// TwinCAT 3 PLC project PLC_Tank
// ProgramVersion: 3.1.4024.0
// libraries:
//   Tc2_ControllerToolbox, * (Beckhoff Automation GmbH)
//   Tc2_ModbusSrv, * (Beckhoff Automation GmbH)
//   Tc2_Standard, * (Beckhoff Automation GmbH)
//   Tc2_System, * (Beckhoff Automation GmbH)
//   Tc3_Module, * (Beckhoff Automation GmbH)
//   VisuDialogs, * (System)
//   VisuSymbols,3.5.10.0,System
// project tree:
//   DUTs/ TAnalogConversion.TcDUT, TEngine.TcDUT, TEngineCmd.TcDUT, THeaterState.TcDUT, THeaterCmd.TcDUT, THeater.TcDUT, TPhaseHeating.TcDUT, TPhaseCmd.TcDUT, TPhaseDraining.TcDUT, TPhaseFilling.TcDUT, TPhaseMixing.TcDUT, TPhaseState.TcDUT, TValveState.TcDUT, TValveCmd.TcDUT, TEngineState.TcDUT, TTank.TcDUT, TValve.TcDUT
//   / GlobalTextList.TcGTLO, PlcTask.TcTTO, PlcTask500ms.TcTTO, Visualization Manager.TcVMO (not stored)
//   GVLs/ Global.TcGVL
//   POUs/ Draining.TcPOU, Engine_1DO.TcPOU, FB_Tank.TcPOU, Filling.TcPOU, Heater.TcPOU, Heating.TcPOU, Main_Batch.TcPOU, MB_Connector.TcPOU, Mixing.TcPOU, Test.TcPOU, Valve_2DO.TcPOU, MAIN.TcPOU
//   POUs/Misc/ EngToRaw.TcPOU, RawToEng.TcPOU
//   VISUs/ Visualization.TcVIS
// real-time tasks:
//   TASK PlcTask: cycle T#100000us, priority 20, ADS port 350
//   TASK PlcTask500ms: cycle T#500ms, priority 1, ADS port 351

CONFIGURATION PLC_Tank
    RESOURCE PLC ON TwinCAT3
        TASK PlcTask(INTERVAL := T#100000us, PRIORITY := 20);
        TASK PlcTask500ms(INTERVAL := T#500ms, PRIORITY := 1);
        PROGRAM MB_Connector WITH PlcTask : MB_Connector;
        PROGRAM Main_Batch WITH PlcTask : Main_Batch;
        PROGRAM MAIN WITH PlcTask500ms : MAIN;
    END_RESOURCE
END_CONFIGURATION

// ---- DUTs/TAnalogConversion.TcDUT
TYPE TAnalogConversion :
STRUCT
	TransducerLoLevel : UINT;
	TransducerHiLevel : UINT;
	ScaledValLoLevel : REAL;
	ScaledValHiLevel : REAL;
END_STRUCT
END_TYPE

// ---- DUTs/TEngine.TcDUT
TYPE TEngine :
STRUCT
	Cmd : TEngineCmd;
	State : TEngineState;
	Time2Start : TIME := T#5S;
	RisingEdgeTrigger : R_TRIG;
	StartupFailTimer : TON;
END_STRUCT
END_TYPE

// ---- DUTs/TEngineCmd.TcDUT
TYPE TEngineCmd :
STRUCT
		SetRT : DINT;
		AutCtrl : BOOL;
		ManCtrl : BOOL;
		TurnOnMan : BOOL;
		TurnOffMan : BOOL;
		Req2RunAutCtrl : BOOL;
		ResetSUF : BOOL;
END_STRUCT
END_TYPE

// ---- DUTs/THeaterState.TcDUT
TYPE THeaterState :
STRUCT
	EnableOut : BOOL;
	HeatingOut : REAL;
	AutCtrl : BOOL;
	ManCtrl : BOOL;
	Err 	: BOOL;
	StateInt : INT;
	GenErr : BOOL; //signalisation: error occured

	HeatingPower : REAL;
	

END_STRUCT
END_TYPE

// ---- DUTs/THeaterCmd.TcDUT
TYPE THeaterCmd :
STRUCT
	AutCtrl : BOOL;
	ManCtrl : BOOL;
	TurnOnMan : BOOL;
	TurnOffMan : BOOL;
	Req2RunAutCtrl : BOOL;
END_STRUCT
END_TYPE

// ---- DUTs/THeater.TcDUT
TYPE THeater :
STRUCT
	Cmd : THeaterCmd;
	State : THeaterState;
	
	ParamHeatingPowerManual : REAL;
	ParamHeatingSetPointAutomat : REAL;
	
	PID : FB_CTRL_PID;
	ThresholdTimer : TON;
	
END_STRUCT
END_TYPE

// ---- DUTs/TPhaseHeating.TcDUT
TYPE TPhaseHeating :
STRUCT
	Cmd : TPhaseCmd;
	State : TPhaseState;
	
	ParamReqTemp : REAL;
	
	WaterTemp : REAL;
	
	fTime : INT;
END_STRUCT
END_TYPE

// ---- DUTs/TPhaseCmd.TcDUT
TYPE TPhaseCmd :
STRUCT
	StartAut : BOOL;
	StopAut : BOOL;
	StartMan : BOOL;
	StopMan : BOOL;
	PauseMan : BOOL;
	ResumeMan : BOOL;
	ResetDone : BOOL;
	AutCtrl : BOOL;
	ManCtrl : BOOL;
END_STRUCT
END_TYPE

// ---- DUTs/TPhaseDraining.TcDUT
TYPE TPhaseDraining :
STRUCT
	Cmd : TPhaseCmd;
	State : TPhaseState;
	
	ParamDrainLevel : REAL;
	WaterLevel : REAL;
END_STRUCT
END_TYPE

// ---- DUTs/TPhaseFilling.TcDUT
TYPE TPhaseFilling :
STRUCT
	Cmd : TPhaseCmd;
	State : TPhaseState;
	
	ParamFillLevel : REAL;
	WaterLevel : REAL;
END_STRUCT
END_TYPE

// ---- DUTs/TPhaseMixing.TcDUT
TYPE TPhaseMixing :
STRUCT
	Cmd : TPhaseCmd;
	State : TPhaseState;
	
	ParamTimeSec : INT;
	
	ElapsedTimeSec : INT;
END_STRUCT
END_TYPE

// ---- DUTs/TPhaseState.TcDUT
TYPE TPhaseState :
STRUCT
	Running : BOOL;
	Idle : BOOL;
	Paused : BOOL;
	Done : BOOL;
	AutCtrl : BOOL;
	ManCtrl : BOOL;
	Stateint : INT;
END_STRUCT
END_TYPE

// ---- DUTs/TValveState.TcDUT
TYPE TValveState :
STRUCT
		Open : BOOL;
		Closed : BOOL;
		OpenOut : BOOL;
		CloseOut : BOOL;
		Err : BOOL;
		StartupFail : BOOL;
		AutCtrl : BOOL;
		ManCtrl : BOOL;
		MayRun : BOOL;
		MayAutoRun : BOOL; //device is working in automatic regime
		GenErr : BOOL; //signalisation: error occured
		StColor : INT; //valve state: Open(0), Closed(1), OpenAndErr(2), ClosedAndErr(3) ,NotOpenNotClosedNotErr(4), NotOpenNotClosedAndErr(5), OpenAndClosedAndErr(6), OpenAndClosedNotErr(7)

END_STRUCT
END_TYPE

// ---- DUTs/TValveCmd.TcDUT
TYPE TValveCmd :
STRUCT
		AutCtrl : BOOL;
		ManCtrl : BOOL;
		OpenMan : BOOL;
		StopMan : BOOL;
		CloseMan : BOOL;
		Req2OpenAut : BOOL;
		Req2CloseAut : BOOL;
		ResetSUF : BOOL;
END_STRUCT
END_TYPE

// ---- DUTs/TEngineState.TcDUT
TYPE TEngineState :
STRUCT
		RT : DINT;
		Run : BOOL;
		RunOut : BOOL;
		Err : BOOL;
		StartUpFail : BOOL;
		AutCtrl : BOOL;
		ManCtrl : BOOL;
		MayRun : BOOL;
		MayAutoRun : BOOL;
		GenErr : BOOL;
		StateInt : INT;
		
		StartupFailTime : INT;
END_STRUCT
END_TYPE

// ---- DUTs/TTank.TcDUT
TYPE TTank :
STRUCT
	Mixer : TEngine;
	ValveFilling : TValve;
	ValveDraining : TValve;
	Heater : THeater;
	
	Filling : TPhaseFilling;
	Draining : TPhaseDraining;
	Mixing : TPhaseMixing;
	Heating : TPhaseHeating;
	
	GlobalError : BOOL;

END_STRUCT
END_TYPE

// ---- DUTs/TValve.TcDUT
TYPE TValve :
STRUCT
	Cmd : TValveCmd;
	State : TValveState;
	Time2Open : TIME := T#12S;
	
	OpenFailTimer : TON;
	CloseFailTimer : TON;
	
END_STRUCT
END_TYPE

// ---- GVLs/Global.TcGVL
{attribute 'qualified_only'}
VAR_GLOBAL
	Tank1 : TTank;
	

	secImp : BOOL;
	
	diMixerRun : BOOL;
	diMixerError : BOOL;
	diValveFillOpen : BOOL;
	diValveFillClose : BOOL;
	diValveFillError : BOOL;
	diValveDrainOpen : BOOL;
	diValveDrainClose : BOOL;
	diValveDrainError : BOOL;
	
	aiWaterLevel : WORD;
	aiWaterTemp : WORD;
	
	doMixerStart : BOOL;
	doValveFillOpen : BOOL;
	doValveFillClose : BOOL;
	doValveDrainOpen : BOOL;
	doValveDrainClose : BOOL;
	doHeatingEnable : BOOL;
	
	aoReqPowerOfHeating : WORD;

END_VAR

VAR_GLOBAL CONSTANT
	Running : INT := 0;
	Stop : INT := 1;
	RunningAndError : INT := 2;
	Err : INT := 3;

	PhIdle : INT := 0;
	PhRunning : INT := 1;
	PhPause : INT := 2;
	
    Open : INT := 0;
	Closed : INT := 1;
	OpenAndErr : INT := 2;
	ClosedAndErr : INT := 3;
	NotOpenNotClosedNotErr : INT := 4;
	NotOpenNotClosedAndErr : INT := 5;
	OpenAndClosedAndErr : INT := 6;
	OpenAndClosedNotErr : INT := 7;
END_VAR

// ---- POUs/MB_Connector.TcPOU
PROGRAM MB_Connector
VAR
	
	mb_ipaddr   : STRING(15) := '127.0.0.1';
	mb_port		: UINT := 503;
	mb_unitid	: BYTE := 1;
	
	fbReadRegs		: FB_MBReadInputRegs;
	mb_regs    		: ARRAY [0..4] OF WORD;
	mb_regs_error	: BOOL;
	mb_regs_busy	: BOOL;
	mb_regs_execute : BOOL;
	mb_regs_errid	: UDINT;
	
	fbReadInps	: FB_MBReadInputs;
	mb_inps			: ARRAY [0..4] OF BYTE;
	mb_inps_error	: BOOL;
	mb_inps_busy	: BOOL;
	mb_inps_execute : BOOL;
	mb_inps_errid	: UDINT;
	
	fbWriteRegs		: FB_MBWriteRegs;
	mbw_regs    	: ARRAY [0..4] OF WORD;
	mbw_regs_error	: BOOL;
	mbw_regs_busy	: BOOL;
	mbw_regs_execute: BOOL;
	mbw_regs_errid	: UDINT;
	
	fbWriteCoils	: FB_MBWriteCoils;
	mbw_coils		: ARRAY [0..4] OF BYTE;
	mbw_coils_error	: BOOL;
	mbw_coils_busy	: BOOL;
	mbw_coils_execute: BOOL;
	mbw_coils_errid	: UDINT;
	
END_VAR

fbReadRegs.sIPAddr := mb_ipaddr;
fbReadRegs.nTCPPort := mb_port;
fbReadRegs.nQuantity := 4;
fbReadRegs.nMBAddr := 0;
fbReadRegs.cbLength := SIZEOF(mb_regs);
fbReadRegs.pDestAddr := ADR(mb_regs);
fbReadRegs.nUnitID := mb_unitid;
fbReadRegs.tTimeout := T#5S;
IF (mb_regs_busy = FALSE) THEN
	mb_regs_execute := TRUE;
ELSE
	mb_regs_execute := FALSE;
END_IF
fbReadRegs(bExecute := mb_regs_execute, 
		   bBusy => mb_regs_busy, bError => mb_regs_error, 
		   nErrId => mb_regs_errid);



fbReadInps.sIPAddr := mb_ipaddr;
fbReadInps.nTCPPort := mb_port;
fbReadInps.nQuantity := 32;
fbReadInps.nMBAddr := 0;
fbReadInps.cbLength := SIZEOF(mb_inps);
fbReadInps.pDestAddr := ADR(mb_inps);
fbReadInps.nUnitID := mb_unitid;
fbReadInps.tTimeout := T#5S;
IF (mb_inps_busy = FALSE) THEN
	mb_inps_execute := TRUE;
ELSE
	mb_inps_execute := FALSE;
END_IF
fbReadInps(bExecute := mb_inps_execute, 
	bBusy => mb_inps_busy, bError => mb_inps_error, nErrId => mb_inps_errid);

Global.diValveFillOpen := mb_inps[0].0;
Global.diValveFillClose := mb_inps[0].1;
Global.diValveFillError := mb_inps[0].2;
Global.diValveDrainOpen := mb_inps[0].3;
Global.diValveDrainClose := mb_inps[0].4;
Global.diValveDrainError := mb_inps[0].5;
Global.diMixerRun := mb_inps[0].6;
Global.diMixerError := mb_inps[0].7;

Global.aiWaterLevel := mb_regs[0];
Global.aiWaterTemp := mb_regs[2];







fbWriteRegs.sIPAddr := mb_ipaddr;
fbWriteRegs.nTCPPort := mb_port;
fbWriteRegs.nQuantity := 4;
fbWriteRegs.nMBAddr := 0;
fbWriteRegs.cbLength := SIZEOF(mbw_regs);
fbWriteRegs.pSrcAddr := ADR(mbw_regs);
fbWriteRegs.nUnitID := mb_unitid;
fbWriteRegs.tTimeout := T#5S;
IF (mbw_regs_busy = FALSE) THEN
	mbw_regs_execute := TRUE;
ELSE
	mbw_regs_execute := FALSE;
END_IF
fbWriteRegs(bExecute := mbw_regs_execute, 
		   bBusy => mbw_regs_busy, bError => mbw_regs_error, 
		   nErrId => mbw_regs_errid);



fbWriteCoils.sIPAddr := mb_ipaddr;
fbWriteCoils.nTCPPort := mb_port;
fbWriteCoils.nQuantity := 32;
fbWriteCoils.nMBAddr := 0;
fbWriteCoils.cbLength := SIZEOF(mbw_coils);
fbWriteCoils.pSrcAddr := ADR(mbw_coils);
fbWriteCoils.nUnitID := mb_unitid;
fbWriteCoils.tTimeout := T#5S;
IF (mbw_coils_busy = FALSE) THEN
	mbw_coils_execute := TRUE;
ELSE
	mbw_coils_execute := FALSE;
END_IF
fbWriteCoils(bExecute := mbw_coils_execute, 
	bBusy => mbw_coils_busy, bError => mbw_coils_error, nErrId => mbw_coils_errid);

mbw_coils[0].0 := Global.doValveFillOpen;
mbw_coils[0].1 := Global.doValveFillClose;
mbw_coils[0].2 := Global.doValveDrainOpen;
mbw_coils[0].3 := Global.doValveDrainClose;
mbw_coils[0].4 := Global.doMixerStart;
mbw_coils[0].5 := Global.doHeatingEnable;

mbw_regs[0] := Global.aoReqPowerOfHeating;

END_PROGRAM

// ---- POUs/Main_Batch.TcPOU
PROGRAM Main_Batch
VAR
	FB_Tank_1 : FB_Tank;
END_VAR

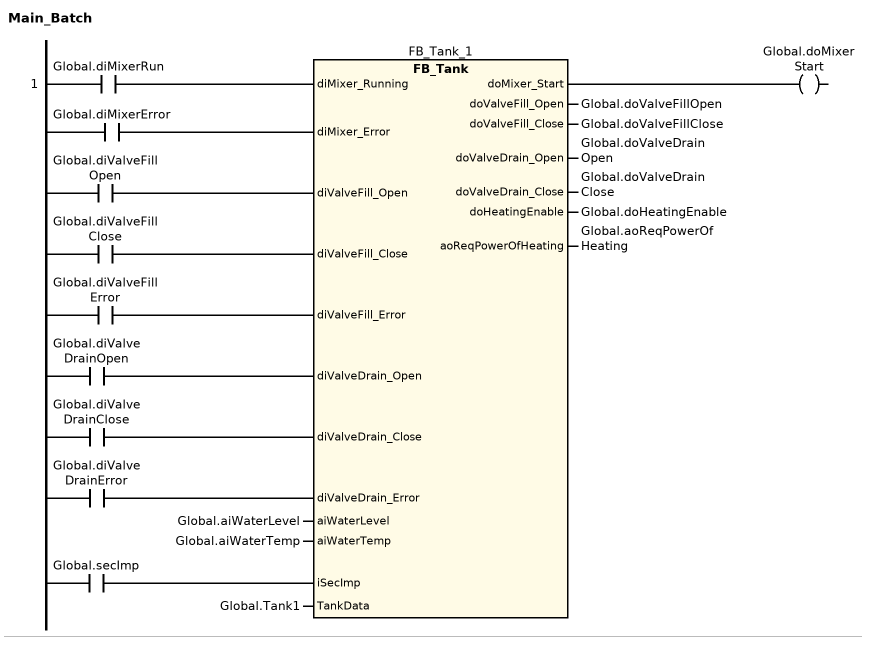
// NETWORK 1
FB_Tank_1(
    diMixer_Running := Global.diMixerRun,
    diMixer_Error := Global.diMixerError,
    diValveFill_Open := Global.diValveFillOpen,
    diValveFill_Close := Global.diValveFillClose,
    diValveFill_Error := Global.diValveFillError,
    diValveDrain_Open := Global.diValveDrainOpen,
    diValveDrain_Close := Global.diValveDrainClose,
    diValveDrain_Error := Global.diValveDrainError,
    aiWaterLevel := Global.aiWaterLevel,
    aiWaterTemp := Global.aiWaterTemp,
    iSecImp := Global.secImp,
    TankData := Global.Tank1,
    doValveFill_Open => Global.doValveFillOpen,
    doValveFill_Close => Global.doValveFillClose,
    doValveDrain_Open => Global.doValveDrainOpen,
    doValveDrain_Close => Global.doValveDrainClose,
    doHeatingEnable => Global.doHeatingEnable,
    aoReqPowerOfHeating => Global.aoReqPowerOfHeating); // FB_Tank
Global.doMixerStart := FB_Tank_1.doMixer_Start;

END_PROGRAM

// ---- POUs/FB_Tank.TcPOU
FUNCTION_BLOCK FB_Tank
VAR_INPUT
	diMixer_Running : BOOL;
	diMixer_Error : BOOL;
	diValveFill_Open : BOOL;
	diValveFill_Close : BOOL;
	diValveFill_Error : BOOL;
	diValveDrain_Open : BOOL;
	diValveDrain_Close : BOOL;
	diValveDrain_Error : BOOL;
	aiWaterLevel : WORD;
	aiWaterTemp : WORD;
	iSecImp : BOOL; //Požaduje se vstup s periodou 1 sekunda a libovolnou střídou
END_VAR

VAR_OUTPUT
	doMixer_Start : BOOL;
	doValveFill_Open : BOOL;
	doValveFill_Close : BOOL;
	doValveDrain_Open : BOOL;
	doValveDrain_Close : BOOL;
	doHeatingEnable : BOOL;
	aoReqPowerOfHeating : WORD;
END_VAR

VAR_IN_OUT
	TankData : TTank;
END_VAR

VAR
	//Konfigurace přepočtu rozsahu převodníků
	WaterTemp : TAnalogConversion := (TransducerLoLevel := 0, TransducerHiLevel := 27648, ScaledValLoLevel := 0, ScaledValHiLevel := 100);
	WaterLevel : TAnalogConversion := (TransducerLoLevel := 0, TransducerHiLevel := 27648, ScaledValLoLevel := 0, ScaledValHiLevel := 2);
	ReqOutputPower : TAnalogConversion := (ScaledValLoLevel := 0, ScaledValHiLevel := 100, TransducerLoLevel := 0, TransducerHiLevel := 27648);

	//Instance zanořených funkčních bloků
	ValveDrainCm : Valve_2DO;
	ValveFillCm : Valve_2DO;
	MixerCm : Engine_1DO;
	HeaterCm : Heater;
	FillingPhase : Filling;
	MixingPhase : Mixing;
	DrainingPhase : Draining;
	HeatingPhase : Heating;
	TON1: TON;
	RawToEng_1: RawToEng;
	RawToEng_2: RawToEng;
	EngToRaw_1: EngToRaw;
END_VAR

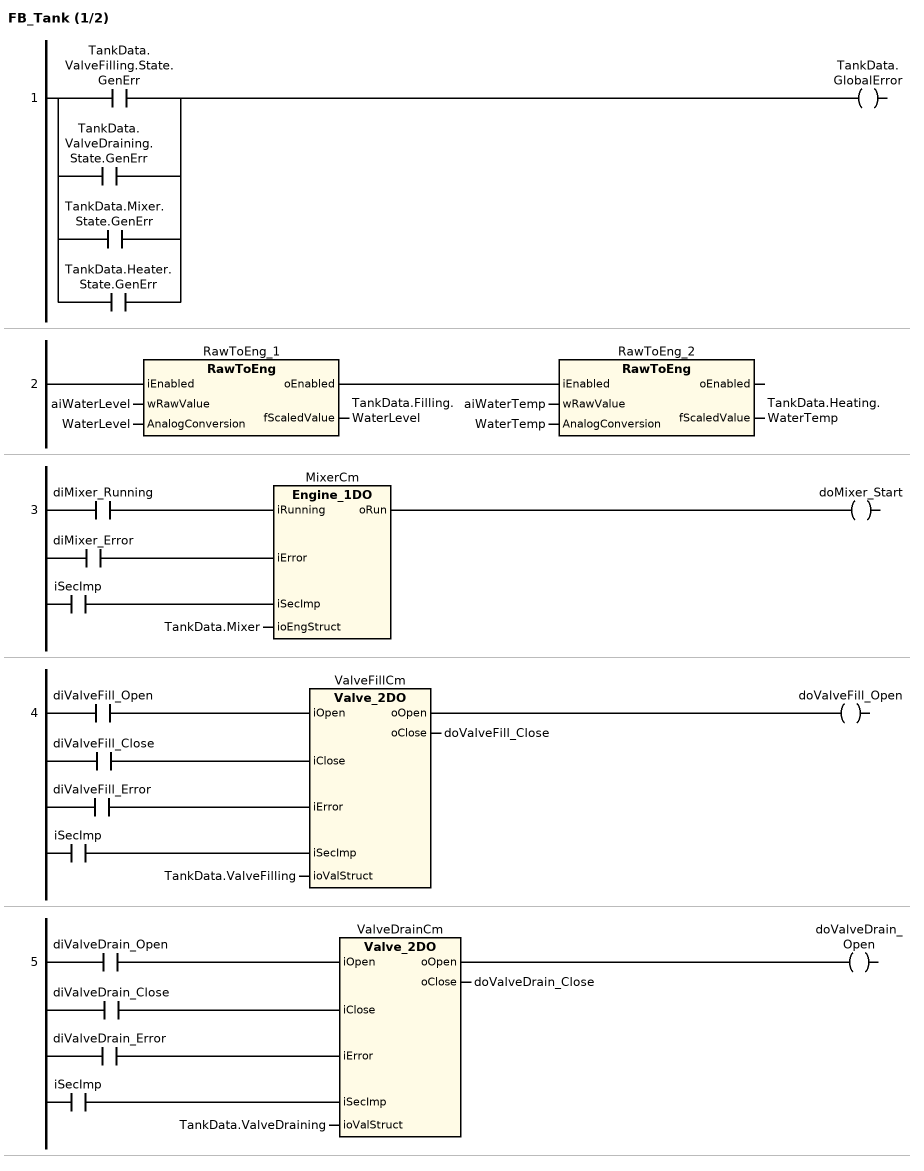
// NETWORK 1
TankData.GlobalError := TankData.ValveFilling.State.GenErr OR TankData.ValveDraining.State.GenErr OR TankData.Mixer.State.GenErr OR TankData.Heater.State.GenErr;

// NETWORK 2
RawToEng_1(
    iEnabled := TRUE,
    wRawValue := aiWaterLevel,
    AnalogConversion := WaterLevel,
    fScaledValue => TankData.Filling.WaterLevel); // RawToEng
RawToEng_2(
    iEnabled := RawToEng_1.oEnabled,
    wRawValue := aiWaterTemp,
    AnalogConversion := WaterTemp,
    fScaledValue => TankData.Heating.WaterTemp); // RawToEng

// NETWORK 3
MixerCm(
    iRunning := diMixer_Running,
    iError := diMixer_Error,
    iSecImp := iSecImp,
    ioEngStruct := TankData.Mixer); // Engine_1DO
doMixer_Start := MixerCm.oRun;

// NETWORK 4
ValveFillCm(
    iOpen := diValveFill_Open,
    iClose := diValveFill_Close,
    iError := diValveFill_Error,
    iSecImp := iSecImp,
    ioValStruct := TankData.ValveFilling,
    oClose => doValveFill_Close); // Valve_2DO
doValveFill_Open := ValveFillCm.oOpen;

// NETWORK 5
ValveDrainCm(
    iOpen := diValveDrain_Open,
    iClose := diValveDrain_Close,
    iError := diValveDrain_Error,
    iSecImp := iSecImp,
    ioValStruct := TankData.ValveDraining,
    oClose => doValveDrain_Close); // Valve_2DO
doValveDrain_Open := ValveDrainCm.oOpen;

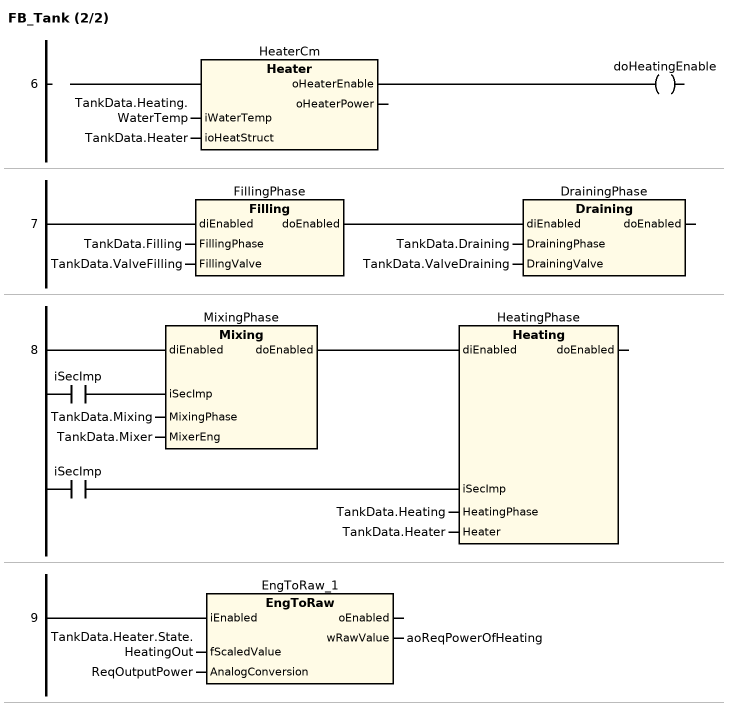
// NETWORK 6
HeaterCm(iWaterTemp := TankData.Heating.WaterTemp, ioHeatStruct := TankData.Heater); // Heater
doHeatingEnable := HeaterCm.oHeaterEnable;

// NETWORK 7
FillingPhase(diEnabled := TRUE, FillingPhase := TankData.Filling, FillingValve := TankData.ValveFilling); // Filling
DrainingPhase(
    diEnabled := FillingPhase.doEnabled,
    DrainingPhase := TankData.Draining,
    DrainingValve := TankData.ValveDraining); // Draining

// NETWORK 8
MixingPhase(
    diEnabled := TRUE,
    iSecImp := iSecImp,
    MixingPhase := TankData.Mixing,
    MixerEng := TankData.Mixer); // Mixing
HeatingPhase(
    diEnabled := MixingPhase.doEnabled,
    iSecImp := iSecImp,
    HeatingPhase := TankData.Heating,
    Heater := TankData.Heater); // Heating

// NETWORK 9
EngToRaw_1(
    iEnabled := TRUE,
    fScaledValue := TankData.Heater.State.HeatingOut,
    AnalogConversion := ReqOutputPower,
    wRawValue => aoReqPowerOfHeating); // EngToRaw

END_FUNCTION_BLOCK

// ---- POUs/Valve_2DO.TcPOU
FUNCTION_BLOCK Valve_2DO
VAR_INPUT
	iOpen : BOOL;
	iClose : BOOL;
	iError : BOOL;
	iSecImp : BOOL;
END_VAR
VAR_OUTPUT
	oOpen : BOOL;
	oClose : BOOL;
END_VAR

VAR_IN_OUT
	ioValStruct	 : TValve;
END_VAR

VAR
	tempOpenStartupFail : BOOL;
	tempCloseStartupFail: BOOL;
END_VAR

{region "OpenState"}
    // set real state of valve input into valve structure - input of valve can be taken from limit sensor...
    ioValStruct.State.Open := iOpen;
    ioValStruct.State.Closed := iClose;
{endregion}

	 
{region "Manual/Automat"}
	// switching state of engine - automatic or manual control (default state is manual)
	
{endregion}
	 
{region "MayRun / MayAutoRun"}
    // setting auxilary signals (may run, may auto run) - MR AND NOT MAR - engine may be started in manual mode, MAR - engine may be started in automatic mode
    ioValStruct.State.MayRun := (ioValStruct.State.ManCtrl AND NOT(ioValStruct.State.GenErr));
	ioValStruct.State.MayAutoRun := (ioValStruct.State.AutCtrl AND NOT(ioValStruct.State.GenErr));
{endregion}
	 
{region "ManCtrl"}
	// processing manual actions - if command is processed, it is sets to FALSE even if can't be processed
    // Valve commands are open, close and stop - valve can be stopped intermediate position
	 IF ioValStruct.State.ManCtrl AND ioValStruct.State.MayRun THEN
        IF ioValStruct.Cmd.OpenMan THEN
            ioValStruct.State.CloseOut := FALSE;
            ioValStruct.State.OpenOut := TRUE;
        END_IF;
        
        IF ioValStruct.Cmd.CloseMan THEN
            ioValStruct.State.OpenOut := FALSE;
            ioValStruct.State.CloseOut := TRUE;
        END_IF;
        
        IF ioValStruct.Cmd.StopMan THEN
            ioValStruct.State.OpenOut := FALSE;
            ioValStruct.State.CloseOut := TRUE;
        END_IF;
    END_IF;
    
    ioValStruct.Cmd.OpenMan := FALSE;
    ioValStruct.Cmd.CloseMan := FALSE;
    ioValStruct.Cmd.StopMan := FALSE;
{endregion}
	 
{region "AutCtrl"}
	 //if request to run in automatic mode -> set outputs to right states if MAR
    //AutoRequest shouldn't be reseted to false state
    //if request to open and request to close are setted to 1 simultaneously - outputs should be 0.
    IF ioValStruct.State.AutCtrl AND ioValStruct.State.MayAutoRun THEN
        IF ioValStruct.Cmd.Req2CloseAut AND (NOT ioValStruct.Cmd.Req2OpenAut) THEN
            ioValStruct.State.OpenOut := FALSE;
            ioValStruct.State.CloseOut := TRUE;
        END_IF;
        
        IF (NOT ioValStruct.Cmd.Req2CloseAut) AND ioValStruct.Cmd.Req2OpenAut THEN
            ioValStruct.State.CloseOut := FALSE;
            ioValStruct.State.OpenOut := TRUE;
        END_IF;
        
        IF (NOT ioValStruct.Cmd.Req2CloseAut) AND (NOT ioValStruct.Cmd.Req2OpenAut) THEN
            ioValStruct.State.CloseOut := FALSE;
            ioValStruct.State.OpenOut := FALSE;
        END_IF;
        
    END_IF;
{endregion}
	 
{region "Error states"}
 // definition of error states 
    // error - input from digital input of plc - fyzical state of valve
    // calculating start up fail - if output is sets to open or close, it's expected feedback from limit sensor in defined time, if feedback doesn't show in this time, it should be start up fail error
    // merge of these two error is general error
    // error is both inputs (open and closed) true state
    ioValStruct.OpenFailTimer(IN := (ioValStruct.State.OpenOut AND (NOT ioValStruct.State.CloseOut)), PT := ioValStruct.Time2Open);
	tempOpenStartupFail := ioValStruct.OpenFailTimer.Q;

    ioValStruct.CloseFailTimer(IN := ((NOT ioValStruct.State.OpenOut) AND ioValStruct.State.CloseOut), PT := ioValStruct.Time2Open);
	tempCloseStartupFail := ioValStruct.CloseFailTimer.Q;
    
   
    IF tempOpenStartupFail OR tempCloseStartupFail THEN
        ioValStruct.State.StartUpFail := TRUE;
    END_IF;
    
    IF iError THEN
        ioValStruct.State.Err := TRUE;
    END_IF;
    
    ioValStruct.State.GenErr := ioValStruct.State.StartUpFail OR iError;
    
    // start up fail can be reseted by operator, command resetSUF, resets SUF and engine should be started again
    IF ioValStruct.Cmd.ResetSUF THEN
        ioValStruct.State.StartUpFail := FALSE;
        ioValStruct.Cmd.ResetSUF := FALSE;
    END_IF;
    
    // if error state exists outputs should be in stop state
    IF ioValStruct.State.GenErr THEN
        ioValStruct.State.OpenOut := FALSE;
        ioValStruct.State.CloseOut := FALSE;
    END_IF;
{endregion}
	 	 
oOpen := ioValStruct.State.OpenOut;
oClose := ioValStruct.State.CloseOut;

{region "StatusInt"}
    //write combination of states into int value for visualization (valve - combination of open, close state and error)
    IF ioValStruct.State.Open AND NOT ioValStruct.State.Closed AND NOT ioValStruct.State.GenErr THEN
        ioValStruct.State.StColor := Global.Open;
    ELSIF NOT ioValStruct.State.Open AND ioValStruct.State.Closed AND NOT ioValStruct.State.GenErr THEN
        ioValStruct.State.StColor := Global.Closed;
    ELSIF ioValStruct.State.Open AND NOT ioValStruct.State.Closed AND ioValStruct.State.GenErr THEN
        ioValStruct.State.StColor := Global.OpenAndErr;
    ELSIF NOT ioValStruct.State.Open AND ioValStruct.State.Closed AND ioValStruct.State.GenErr THEN
        ioValStruct.State.StColor := Global.ClosedAndErr;
    ELSIF NOT ioValStruct.State.Open AND NOT ioValStruct.State.Closed AND NOT ioValStruct.State.GenErr THEN
        ioValStruct.State.StColor := Global.NotOpenNotClosedNotErr;
    ELSIF NOT ioValStruct.State.Open AND NOT ioValStruct.State.Closed AND ioValStruct.State.GenErr THEN
        ioValStruct.State.StColor := Global.NotOpenNotClosedAndErr;
    ELSIF ioValStruct.State.Open AND ioValStruct.State.Closed AND ioValStruct.State.GenErr THEN
        ioValStruct.State.StColor := Global.OpenAndClosedAndErr;
    ELSIF ioValStruct.State.Open AND ioValStruct.State.Closed AND NOT ioValStruct.State.GenErr THEN
        ioValStruct.State.StColor := Global.OpenAndClosedNotErr;
    END_IF;
{endregion}

END_FUNCTION_BLOCK

// ---- POUs/Engine_1DO.TcPOU
FUNCTION_BLOCK Engine_1DO
VAR_INPUT
	iRunning : BOOL;
	iError : BOOL;
	iSecImp : BOOL;
END_VAR
VAR_OUTPUT
	oRun : BOOL;
END_VAR
VAR_IN_OUT
	ioEngStruct : TEngine;
END_VAR
VAR
	secImpEdge: BOOL;
	tempStartupFail: BOOL;
END_VAR

{region "RunState"}
    // set real state of engine run into engine structure
  
{endregion}

{region "Running time"} 
    // counting running time of engine - (motoseconds in real situation it should be moto hours)
    // detection rising edge of input secimp - should be conected 1Hz internal clock from PLC
	
{endregion}
	 
 
{region "Manual/Automat"}
	// switching state of engine - automatic or manual control (default state is manual)
	
{endregion}
	 
{region "MayRun / MayAutoRun"}
	// setting auxilary signals (may run, may auto run) - MR AND NOT MAR - eng should be started in manual mode,
    // MAR - should be started in automatic mode
    ioEngStruct.State.MayRun := (ioEngStruct.State.ManCtrl AND NOT(ioEngStruct.State.GenErr));
	ioEngStruct.State.MayAutoRun := (ioEngStruct.State.AutCtrl AND NOT(ioEngStruct.State.GenErr));
		 
			  
{endregion}
	 
{region "ManCtrl"}
	// processing manual actions - if command is processed, it is set to FALSE even if can't be processed
    // Engine commands are turn off (stop) and turn on (start)
	
{endregion}
	 
{region "AutCtrl"}
	//if request to run in automatic mode set outputs to right states if MAR
    //AutoRequest shouldn't be reseted to false state
    
{endregion}
	 
{region "Error states"}
	// definition of error states 
	// error - input from digital input of plc - fyzical state of engine 
	// calculating start up fail - if output is sets to start engine, it's expected feedback from running signal in defined time, if feedback doesn't show in this time, it should be start up fail error
	// merge of these two error is general error
	
{endregion}
	 
oRun := ioEngStruct.State.RunOut;

{region "StatusInt"}
 IF NOT ioEngStruct.State.GenErr THEN
        IF ioEngStruct.State.Run THEN
            ioEngStruct.State.StateInt := Global.Running;
        ELSE
            ioEngStruct.State.StateInt := Global.Stop;
        END_IF;
    ELSE
        IF ioEngStruct.State.Run THEN
            ioEngStruct.State.StateInt := Global.RunningAndError;
        ELSE
            ioEngStruct.State.StateInt := Global.Err;
        END_IF;
    END_IF; 
{endregion}

END_FUNCTION_BLOCK

// ---- POUs/Heater.TcPOU
FUNCTION_BLOCK Heater
VAR_INPUT
	iWaterTemp : REAL;
END_VAR
VAR_OUTPUT
	oHeaterEnable : BOOL;
	oHeaterPower : REAL;
END_VAR
VAR_IN_OUT
	ioHeatStruct : THeater;
END_VAR
VAR
	pidParameters : ST_CTRL_PID_PARAMS;
END_VAR

pidParameters.fKp := 10; //P
pidParameters.tTn := T#2S; //I
pidParameters.tTv := T#0.5S; //D
pidParameters.tCtrlCycleTime := T#200MS;
pidParameters.tTaskCycleTime := T#100MS;
pidParameters.fOutMaxLimit := 100;
pidParameters.fOutMinLimit := 0;
pidParameters.bDInTheFeedbackPath := FALSE;
pidParameters.bPInTheFeedbackPath := FALSE;
pidParameters.bARWOnIPartOnly := FALSE;
pidParameters.tTd := T#100MS; 

ioHeatStruct.PID(
	fSetpointValue := ioHeatStruct.ParamHeatingSetPointAutomat, 
	fActualValue := iWaterTemp, 
	fManSyncValue := ioHeatStruct.ParamHeatingPowerManual,
	bSync := ioHeatStruct.State.ManCtrl,
	eMode := E_CTRL_MODE.eCTRL_MODE_ACTIVE, // automatic mode of PID component
	stParams := pidParameters);

ioHeatStruct.State.HeatingOut := ioHeatStruct.PID.fOut;

	 
{region "Manual/Automat"}
// switching state of engine - automatic or manual control (default state is manual)

{endregion}
	 
 
{region "ManCtrl"}
// processing manual actions - if command is processed, it is set to FALSE even if can't be processed
// Engine commands are turn off (stop) and turn on (start)

{endregion}
 
{region "AutCtrl"}
//if request to run in automatic mode set outputs to right states if MAR
//AutoRequest shouldn't be reseted to false state

{endregion}
 
{region "Error states"}
// if water temperature is too high, stop heating and generate error

{endregion}
	 
 
oHeaterPower := ioHeatStruct.State.HeatingOut;
oHeaterEnable := ioHeatStruct.State.EnableOut;

END_FUNCTION_BLOCK

// ---- POUs/Filling.TcPOU
FUNCTION_BLOCK Filling
VAR_INPUT
    diEnabled : BOOL; // Aktivace fáze
END_VAR
VAR_OUTPUT
    doEnabled : BOOL; // Výstupní povolení fáze
END_VAR
VAR_IN_OUT
    FillingPhase : TPhaseFilling; // Struktura fáze napouštění
    FillingValve : TValve;       // Struktura ventilu
END_VAR
VAR
    isManual : BOOL; // Příznak manuálního režimu
END_VAR


{region "REGION Aut/Man"}
// Přepínání mezi režimy
IF FillingPhase.Cmd.ManCtrl THEN
    isManual := TRUE;
    FillingPhase.State.ManCtrl := TRUE;
    FillingPhase.State.AutCtrl := FALSE;
ELSE
    isManual := FALSE;
    FillingPhase.State.ManCtrl := FALSE;
    FillingPhase.State.AutCtrl := TRUE;
END_IF;
{endregion}

{region "ManCtrl"}
// Manuální režim
IF isManual THEN
    IF FillingPhase.Cmd.StartMan THEN
        FillingValve.Cmd.OpenMan := TRUE;
        FillingPhase.State.Running := TRUE;
        FillingPhase.Cmd.StartMan := FALSE;
    END_IF;

    IF FillingPhase.Cmd.StopMan OR FillingPhase.Cmd.PauseMan THEN
        FillingValve.Cmd.CloseMan := TRUE;
        FillingPhase.State.Running := FALSE;
        FillingPhase.Cmd.StopMan := FALSE;
        FillingPhase.Cmd.PauseMan := FALSE;
    END_IF;

    IF FillingPhase.Cmd.ResumeMan THEN
        FillingValve.Cmd.OpenMan := TRUE;
        FillingPhase.State.Running := TRUE;
        FillingPhase.Cmd.ResumeMan := FALSE;
    END_IF;
END_IF;
{endregion}

{region "AutCtrl"}
// Automatický režim
IF NOT isManual THEN
    IF FillingPhase.WaterLevel < FillingPhase.ParamFillLevel THEN
        FillingValve.Cmd.Req2OpenAut := TRUE;
        FillingValve.Cmd.Req2CloseAut := FALSE;
        FillingPhase.State.Running := TRUE;
    ELSE
        FillingValve.Cmd.Req2OpenAut := FALSE;
        FillingValve.Cmd.Req2CloseAut := TRUE;
        FillingPhase.State.Running := FALSE;
    END_IF;
END_IF;
{endregion}

{region "Done"}
// Podmínka dokončení
IF FillingPhase.WaterLevel >= FillingPhase.ParamFillLevel THEN
    FillingPhase.State.Done := TRUE;
    FillingPhase.State.Running := FALSE;
    FillingValve.Cmd.Req2CloseAut := TRUE;
END_IF;
{endregion}

// Povolení fáze
doEnabled := diEnabled;

END_FUNCTION_BLOCK

// ---- POUs/Mixing.TcPOU
FUNCTION_BLOCK Mixing
VAR_INPUT
	diEnabled : BOOL;
	iSecImp : BOOL;
END_VAR
VAR_OUTPUT
	doEnabled : BOOL;
END_VAR
VAR_IN_OUT
	MixingPhase : TPhaseMixing;
	MixerEng : TEngine;
END_VAR
VAR
END_VAR

{region "Aut/Man"}
    // switching state of engine - automatic or manual control (default state is manual)
  
{endregion}

{region "ManCtrl"}
    // processing manual actions - if command is processed, it is sets to FALSE even if can't be processed
    // Phase commands are start, stop, pause and resume 
    // Start - start mixing  
    // Stop - stop mixing
    // Pause - stop mixing 
    // Resume - start mixing
    // real states of phase are writed into states in phase structure
   
{endregion}

{region "AutCtrl"}
    // if request to run in automatic mode -> set auto request to mixing to 1, if not request to mixing is 0
    // commands should be sets to false after their processing
   
{endregion}

{region "Done"}
    // every phase should have finish condition - mixing phase - if time of runnig is bigger or same as requested
    // after that done state should be setted to 1
 
{endregion}

{region "States"}
    //Command mixer in cases of states

{endregion}
 MixingPhase.State.Running := TRUE;

// delault state of phase - if not any state sets state to idle
IF NOT MixingPhase.State.Idle AND NOT MixingPhase.State.Done AND NOT MixingPhase.State.Paused AND NOT MixingPhase.State.Running THEN
    MixingPhase.State.Idle := 1;
END_IF;


// delault state of phase - if not any state sets state to idle
IF MixingPhase.State.Idle THEN
    MixingPhase.State.StateInt := Global.PhIdle;
ELSIF MixingPhase.State.Running THEN
    MixingPhase.State.StateInt := Global.PhRunning;
ELSE
    MixingPhase.State.StateInt := Global.PhPause;
END_IF;

doEnabled := diEnabled;

END_FUNCTION_BLOCK

// ---- POUs/Draining.TcPOU
FUNCTION_BLOCK Draining
VAR_INPUT
	diEnabled : BOOL;
END_VAR
VAR_OUTPUT
	doEnabled : BOOL;
END_VAR
VAR_IN_OUT
	DrainingPhase : TPhaseDraining;
	DrainingValve : TValve;
END_VAR
VAR
END_VAR

{region "Aut/Man"}
    // switching state of engine - automatic or manual control (default state is manual)
  
{endregion}

{region "ManCtrl"}
    // processing manual actions - if command is processed, it is sets to FALSE even if can't be processed
    // Phase commands are start, stop, pause and resume 
    // Start - open draining valve 
    // Stop - close draining valve
    // Pause - close draining valve
    // Resume - open draining valve
    // real states of phase are writed into states in phase structure
  
{endregion}

{region "AutCtrl"}
    //if request to run in automatic mode -> set auto request to open of filling valve to 1 and close to 0, if not open 0 close 1
    // commands should be sets to false after their processing
   
{endregion}
{region "Done"}
    //every phase should have finish condition - draining phase - if water level is below requested level
    //after that done state should be setted to 1
   
{endregion}

{region "States"} 
    //Command valve in cases of states
   
{endregion}

// delault state of phase - if not any state sets state to idle
IF (NOT DrainingPhase.State.Idle) AND (NOT DrainingPhase.State.Paused) AND (NOT DrainingPhase.State.Running) THEN
    DrainingPhase.State.Idle := 1;
END_IF;

// write binary states into int value for visualization
IF DrainingPhase.State.Idle THEN
    DrainingPhase.State.StateInt := Global.PhIdle;
ELSIF DrainingPhase.State.Running THEN
    DrainingPhase.State.StateInt := Global.PhRunning;
ELSE
    DrainingPhase.State.StateInt := Global.PhPause;
END_IF;

//Ponechte pro moznost retezeni volani bloku v LAD
doEnabled := diEnabled;

END_FUNCTION_BLOCK

// ---- POUs/Heating.TcPOU
FUNCTION_BLOCK Heating
VAR_INPUT
	diEnabled : BOOL;
	iSecImp : BOOL;
END_VAR
VAR_OUTPUT
	doEnabled : BOOL;
END_VAR
VAR_IN_OUT
	HeatingPhase : TPhaseHeating;
	Heater : THeater;
END_VAR
VAR
	pidParameters : ST_CTRL_PID_PARAMS;
END_VAR

{region "Aut/Man"}
    // switching state of engine - automatic or manual control (default state is manual)
 
{endregion}

{region "ManCtrl"}
    // processing manual actions - if command is processed, it is sets to FALSE even if can't be processed
        // real states of phase are writed into states in phase structure
    
   
{endregion}

{region "AutCtrl"}
    // if request to run in automatic mode -> set auto request to heat to 1, if not request to heat 0
    // commands should be sets to false after their processing
  
{endregion}

{region "Done"}
    //every phase should have finish condition - heating phase - if water temp is on requested value for 15 seconds with 1°C hysteresis
    //after that done state should be setted to 1



    // command reset done resets done state and than resets command
  
{endregion}

{region "States"}
    //Command valve in cases of states
    // Running - start heating  
    // Idle - stop heating
    // Pause - stop heating (alternative is hold actual temp)
  
{endregion}

// delault state of phase - if not any state sets state to idle
IF NOT HeatingPhase.State.Idle AND NOT HeatingPhase.State.Paused AND NOT HeatingPhase.State.Running THEN
    HeatingPhase.State.Idle := 1;
END_IF;

doEnabled := diEnabled;

END_FUNCTION_BLOCK

// ---- POUs/Misc/RawToEng.TcPOU
FUNCTION_BLOCK RawToEng
VAR_INPUT
	iEnabled : BOOL;
	wRawValue : WORD;
	AnalogConversion : TAnalogConversion;
END_VAR
VAR_OUTPUT
	oEnabled : BOOL;
	fScaledValue : REAL;
END_VAR
VAR
END_VAR

//Prepocet z wRawValue (z procesu po ModbusTCP) na fScaledValue (do PLC) podle parametru v AnalogConversion.

//Filtrace hodnoty, bylo by vhodne odfiltrovat take kmitani z minimalniho rozsahu na maximalni hodnotu 27648
IF wRawValue = 27648 THEN 
	wRawValue := 0; //Ale lepe nez takto...
END_IF

fScaledValue:= (AnalogConversion.ScaledValHiLevel-AnalogConversion.ScaledValLoLevel) * (wRawValue-AnalogConversion.TransducerLoLevel)/(AnalogConversion.TransducerHiLevel-AnalogConversion.TransducerLoLevel) + AnalogConversion.ScaledValLoLevel;
oEnabled := iEnabled;

END_FUNCTION_BLOCK

// ---- POUs/Misc/EngToRaw.TcPOU
FUNCTION_BLOCK EngToRaw
VAR_INPUT
	iEnabled : BOOL;
	fScaledValue : REAL;
	AnalogConversion : TAnalogConversion;
END_VAR
VAR_OUTPUT
	oEnabled : BOOL;
	wRawValue : WORD;
END_VAR
VAR
END_VAR

//Prepocet z fScaledValue (z PLC) na wRawValue (do procesu po ModbusTCP) podle parametru v AnalogConversion.
wRawValue := REAL_TO_WORD((AnalogConversion.TransducerHiLevel - AnalogConversion.TransducerLoLevel) * (fScaledValue - AnalogConversion.ScaledValLoLevel) / (AnalogConversion.ScaledValHiLevel - AnalogConversion.ScaledValLoLevel) + AnalogConversion.TransducerLoLevel);
oEnabled := iEnabled;

END_FUNCTION_BLOCK

// ---- POUs/MAIN.TcPOU
PROGRAM MAIN
VAR
    // Instance funkčního bloku Filling
    fbFilling : Filling;

    // Struktura fáze Filling
    fillingPhase : TPhaseFilling;

    // Struktura ventilu
    fillingValve : TValve;

    // Globální časový impuls
    secImp : BOOL;

    isManual : BOOL; // Manuální režim
END_VAR

// Generování časového impulsu
Global.secImp := NOT(Global.secImp);

// Nastavení režimu (příklad pro testování)
isManual := TRUE; // Přepínání mezi manuálním a automatickým režimem

END_PROGRAM

// ---- POUs/Test.TcPOU
PROGRAM Test
VAR
	State : INT := 0;
END_VAR

CASE State OF
	1:  Global.Tank1.Filling.ParamFillLevel := 1.8;
		Global.Tank1.Filling.Cmd.ManCtrl := TRUE;
		Global.Tank1.Filling.Cmd.StartMan:= TRUE;
		IF Global.Tank1.Filling.State.Done = TRUE THEN
			State := 2;
		END_IF
	2: //...
END_CASE

END_PROGRAM

// ---- GlobalTextList.TcGTLO
TEXTLIST GlobalTextList
  815 = 'ABC'
  406 = 'AUT'
  473 = 'Checkbox'
  70 = 'Close'
  25 = 'Closed'
  201 = 'Filling Valve'
  560 = 'MAN'
  604 = 'Open'
  687 = 'Opened'
  98 = 'Res. SUF'
  256 = 'SUF'
END_TEXTLIST

// ---- VISUs/Visualization.TcVIS
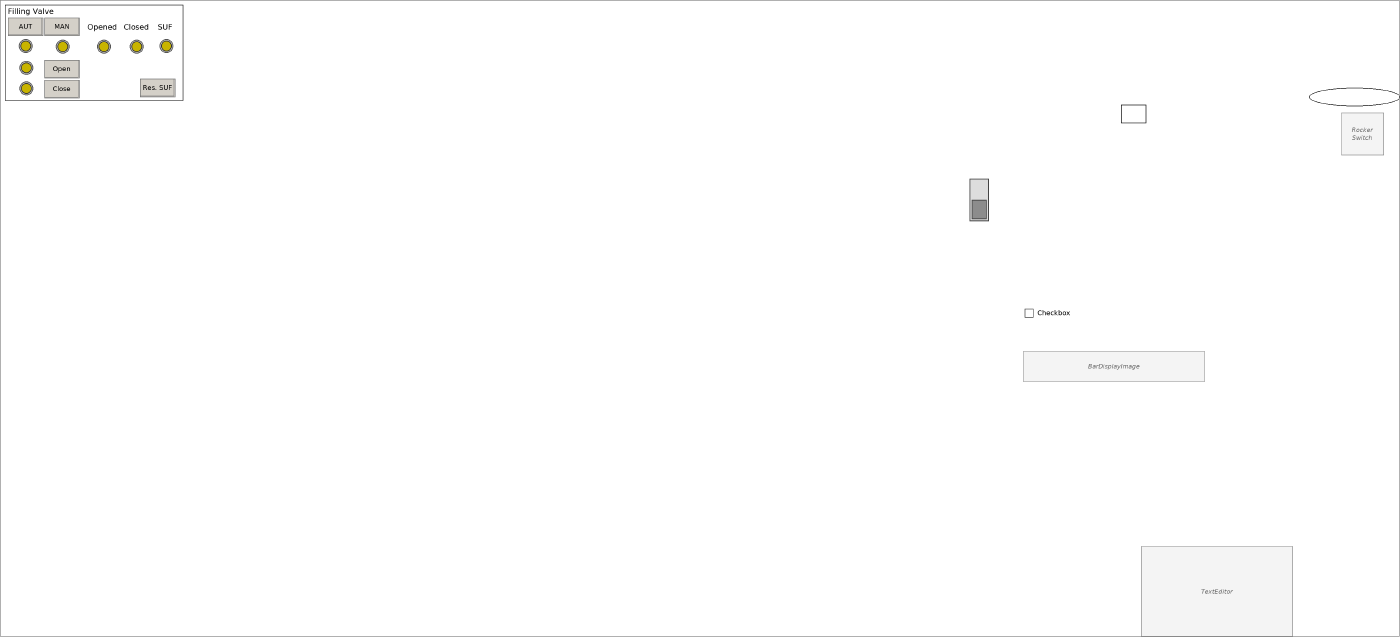
VISUALIZATION Visualization  // 2309x1052
    Rectangle (8,8 294x158)
    Checkbox (1688,502 150x30), "Checkbox"
    BarDisplayImage (1687,580 300x50), style: BarDisplayImage-Gray, scale format: %.1f, scale 0..100
    DipSwitch (1580,295 70x70), behaviour: TOGGLE, style: Switch-DipSwitch-Gray
    RockerSwitch (2212,186 70x70), behaviour: TOGGLE, style: Switch-RockerSwitch-Gray
    TextEditor (1882,902 250x150)
        p4127561890: Courier New
    Ellipse (2159,145 150x30)
    Rectangle (1849,173 41x30)
    Button (13,29 58x30), "AUT"
        OnMouseClick: toggle Global.Tank1.ValveFilling.Cmd.AutCtrl
    Button (73,29 58x30), "MAN"
        OnMouseClick: toggle Global.Tank1.ValveFilling.Cmd.ManCtrl
    Label (10,10 96x18), "Filling Valve"
    Button (73,99 58x30), "Open"
        OnMouseClick: toggle Global.Tank1.ValveFilling.Cmd.OpenMan
    Button (73,132 58x30), "Close"
        OnMouseClick: toggle Global.Tank1.ValveFilling.Cmd.CloseMan
    Lamp1 (29,63 27x26), variable: Global.Tank1.ValveFilling.State.AutCtrl, style: Lamp-Lamp1-Yellow
    Lamp1 (90,64 27x26), variable: Global.Tank1.ValveFilling.State.ManCtrl, style: Lamp-Lamp1-Yellow
    Lamp1 (158,64 27x26), variable: Global.Tank1.ValveFilling.State.Open, style: Lamp-Lamp1-Yellow
    Lamp1 (212,64 27x26), variable: Global.Tank1.ValveFilling.State.Closed, style: Lamp-Lamp1-Yellow
    Lamp1 (261,63 27x26), variable: Global.Tank1.ValveFilling.State.StartupFail, style: Lamp-Lamp1-Yellow
    Button (231,130 58x30), "Res. SUF"
        OnMouseClick: toggle Global.Tank1.ValveFilling.Cmd.ResetSUF
    Label (141,36 53x18), "Opened"
    Label (201,36 53x18), "Closed"
    Label (257,36 33x18), "SUF"
    Lamp1 (30,99 27x26), variable: Global.Tank1.ValveFilling.State.OpenOut, style: Lamp-Lamp1-Yellow
    Lamp1 (30,133 27x26), variable: Global.Tank1.ValveFilling.State.CloseOut, style: Lamp-Lamp1-Yellow
END_VISUALIZATION
